Staubli VAL3: AdjustTraj.pgx

public program AdjustTraj(num x_nTrajIndex)
  local bool l_bRes
  local num l_nNum
begin


  //调图主界面，入口

  cls()

  call UI:Control_PanelMd("请等待，正在读取文件......")
  TxtFile:bStartRead=true
  DataBase:bStopPoll=true

  //删除临时文件
  if $fileExists("Disk://Txt/1.txt")
    $delete("Disk://Txt/1.txt")
  endIf

  if $fileExists("Disk://Txt/2.txt")
    $delete("Disk://Txt/2.txt")
  endIf

  if $fileExists("Disk://Txt/3.txt")
    $delete("Disk://Txt/3.txt")
  endIf

  if $fileExists("Disk://Txt/4.txt")
    $delete("Disk://Txt/4.txt")
  endIf




  call TxtFile:IsAdjustTraj("Disk://Txt/Recipe.txt",TxtFile:sProductName,x_nTrajIndex,x_nTrajIndex,l_bRes)
  call TxtFile:CloseFile()
  if !l_bRes
    DataBase:bStopPoll=false
    popUpMsg("文件读取出错!")
    return
  endIf


  //参数初始化
  bFirstTeach=true
  DataBase:bStopPoll=false
  //路径界面
  call TrajScreen()


end
